INTERFACE ITF_BaseMainComponent

END_INTERFACE

(* stored: Version 1.1.0.1
   Itf ITF_BaseMainComponent: Id {2822f205-b986-005f-04be-ccc64a012929} *)
